# EPICS autosave request: iocs/rixscamIOC/iocBoot/iocRixsCam/auto_settings.req
file "xcamCamera_settings.req",    P=$(P),  R=Camera1:
file "NDStdArrays_settings.req",    P=$(P), R=image1:
file "NDPluginXIP_settings.req",	P=$(P),	R=XIP1:
file "commonPluginsLocal_settings.req",   P=$(P)
